// TwinCAT 3 PLC project PLC
// Title: Spreizanlage
// Company: fhnw
// ProjectVersion: 1.0.0.0
// ProgramVersion: 3.1.4026.14
// CompilerDefines: VISU_USEPROPERTYINFO
// libraries:
//   Tc2_MC2, * (Beckhoff Automation GmbH)
//   Tc2_Standard, * (Beckhoff Automation GmbH)
//   Tc2_System, * (Beckhoff Automation GmbH)
//   Tc2_TcpIp, * (Beckhoff Automation GmbH)
//   Tc2_Utilities, * (Beckhoff Automation GmbH)
//   VisuDialogs, * (System)
//   VisuSymbols, * (System)
// project tree:
//   DUTs/ ProcessData.TcDUT, State.TcDUT
//   / GlobalTextList.TcGTLO, PlcTask.TcTTO, Visualization Manager.TcVMO (not stored), VISU_TASK.TcTTO
//   GVLs/ GVL.TcGVL, GVL_Axis.TcGVL, GVL_HMI.TcGVL, GVL_Parameter.TcGVL
//   Lib/UDP/ FB_UDP_Connection.TcPOU, FB_UDP_ScanControl30x0.TcPOU
//   POUs/ FB_ControlPad.TcPOU, FB_FileWriter.TcPOU, FB_Izumi.TcPOU, FB_LaserScanner.TcPOU, FB_Winder.TcPOU, MAIN.TcPOU
//   VISUs/ GeneralSettings.TcVIS, MainWindow.TcVIS, Manual_Mode.TcVIS, Production_Mode.TcVIS, Setup_Mode.TcVIS, Winder_control.TcVIS
// real-time tasks:
//   TASK PlcTask: cycle T#10ms, priority 20, ADS port 350
//   TASK VisuTask: cycle T#200000us, priority 30, ADS port 351
// motion (NC):
//   TASK NC-Task 1 SAF: cycle T#2ms, priority 4, ADS port 501
//   TASK NC-Task 1 SVB: cycle T#10ms, priority 8, ADS port 511
//   AXIS Achse 1 (id 1)
//     General: UnitName=°
//     Dynamic: Acceleration=1592.706, Deceleration=1592.706, Jerk=4778.118
//     Velo: RefSearch=10.61804, RefSync=10.61804, SlowManual=53.0902, FastManual=318.5412, Fast=1061.804, Maximum=1061.804
//     OtherSettings: AllowMotionCmdToSlave=true
//     encoder EncType=19
//       EncPara: ScaleFactorNumerator=360, ScaleFactorDenominator=12582912, Inverse=true, MaxCount=#xffffffff
//     drive DrvType=16
//       DrvPara: Inverse=true, MaxCount=#xffffffff, DriveControlDWord=#x00020000
//         Analog: VeloReferenz=1167.9844, VeloScale=32, TorqueSetpointScale=10, ScaleFactorActTorque=0.1
//         TimeComp: TaskDelayCycles=1
//     controller CtrType=1
//       CtrPara: PriorControlFactor=1
//         Observer: BandWidth=20
// I/O:
//   DEVICE Gerät 1 (EtherCAT), AmsNetId 192.168.1.15.2.1
//     Klemme 1 (EK1100) [EK1100 EtherCAT-Koppler (2A E-Bus)]
//       Klemme 2 (EL1859) [EL1859 8K. Dig. Eingang 24V, 3ms, 8K. Dig. Ausgang 24V, 0.5A]
//       Klemme 3 (EL3064) [EL3064 4K.Ana. Eingang 0-10V]
//       Klemme 4 (ELM7221-0010) [ELM7221-0010 1K. Servo-Motor-Endstufe (48 V, 8 A RMS OCT)]
//         startup 32785:27 := E02E0000 // DRV Motor Settings Ch.1 / Motor speed limitation
//         startup 28688:3 := 08 // DRV Outputs Ch.1 / Modes of operation
//         startup 28688:16 := FF7F // DRV Outputs Ch.1 / Positive torque limit value
//         startup 28688:17 := FF7F // DRV Outputs Ch.1 / Negative torque limit value
//         startup 32784:87 := 64 // DRV Amplifier Settings Ch.1 / Position loop velocity feed forward gain
//         startup 32784:109 := 64000000 // DRV Amplifier Settings Ch.1 / Torque feed forward gain
//         startup 28688:11 := A00F // DRV Outputs Ch.1 / Torque limitation
//         startup 32784:19 := 2C02 // DRV Amplifier Settings Ch.1 / Current loop proportional gain
//         startup 32784:18 := 1500 // DRV Amplifier Settings Ch.1 / Current loop integral time
//         startup 32784:21 := 70000000 // DRV Amplifier Settings Ch.1 / Velocity loop proportional gain
//         startup 32784:20 := 96000000 // DRV Amplifier Settings Ch.1 / Velocity loop integral time
//       Klemme 5 (EL2634) [EL2634 4K. Relais Ausgang, Schließer (250 AC / 30V DC)]
//       Klemme 7 (EL9011) [EL9011 Endklemme]
//     Box 6 (NETX 51-RE/ECS) [NETX 51-RE/ECS]
// variable links:
//   NC-Task 1 SAF/Axes/Achse 1 <-> Device 1 (EtherCAT)/Term 1 (EK1100)/Term 4 (ELM7221-0010)
//     Drive/Inputs/In/nDataIn1 <-> DRV Following error actual value/Following error actual value
//     Drive/Inputs/In/nDataIn3[0] <-> DRV Torque actual value/Torque actual value
//     Drive/Inputs/In/nDcOutputTime <-> InfoData/DcOutputShift
//     Drive/Inputs/In/nState1 <-> DRV Statusword/Statusword
//     Drive/Inputs/In/nState2 <-> DRV Statusword/Statusword @bit 8
//     Drive/Inputs/In/nState4 @bit 1 <-> WcState/InputToggle
//     Drive/Inputs/In/nState4 <-> WcState/WcState
//     Drive/Outputs/Out/nCtrl1 <-> DRV Controlword/Controlword
//     Drive/Outputs/Out/nCtrl2 <-> DRV Controlword/Controlword @bit 8
//     Drive/Outputs/Out/nDataOut1 <-> DRV Target position/Target position
//     Drive/Outputs/Out/nDataOut2 <-> DRV Target velocity/Target velocity
//     Enc/Inputs/In/nDataIn1 <-> FB Position/Position
//     Enc/Inputs/In/nDcInputTime <-> InfoData/DcInputShift
//     Enc/Inputs/In/nState4 @bit 1 <-> WcState/InputToggle
//     Enc/Inputs/In/nState4 <-> WcState/WcState
//   PLC Instance <-> Device 1 (EtherCAT)/Term 1 (EK1100)/Term 2 (EL1859)
//     PlcTask Inputs/MAIN.ControlPad.bDigital_DecSpeed <-> Channel 5/Input
//     PlcTask Inputs/MAIN.ControlPad.bDigital_EStop <-> Channel 1/Input
//     PlcTask Inputs/MAIN.ControlPad.bDigital_IncSpeed <-> Channel 4/Input
//     PlcTask Inputs/MAIN.ControlPad.bDigital_Start <-> Channel 3/Input
//     PlcTask Inputs/MAIN.ControlPad.bDigital_Stop <-> Channel 2/Input
//   PLC Instance <-> Device 1 (EtherCAT)/Term 1 (EK1100)/Term 3 (EL3064)
//     PlcTask Inputs/MAIN.fbIzumi.iIzumiData <-> AI Standard Channel 1/Value
//   PLC Instance <-> NC-Task 1 SAF/Axes/Achse 1
//     PlcTask Inputs/MAIN.fbWinder.winderAxis.NcToPlc <-> Outputs/ToPlc
//     PlcTask Outputs/MAIN.fbWinder.winderAxis.PlcToNc <-> Inputs/FromPlc

CONFIGURATION PLC
    RESOURCE PLC ON TwinCAT3
        TASK PlcTask(INTERVAL := T#10ms, PRIORITY := 20);
        TASK VISU_TASK(INTERVAL := T#200000us, PRIORITY := 30);
        PROGRAM MAIN WITH PlcTask : MAIN;
        PROGRAM VisuElems_Visu_Prg WITH VISU_TASK : VisuElems.Visu_Prg;
    END_RESOURCE
END_CONFIGURATION

// ---- DUTs/ProcessData.TcDUT
TYPE ProcessData :
STRUCT
    Id          	: DINT;
    Value       	: DINT;
	RunningLength 	: REAL;  // Tape running length [m]
	Torque			: REAL; // Torque [?]
	TapeWidth		: REAL; // Measured width of tape (Laserscanner)
	LateralGap		: REAL;
	Airflow			: REAL;
	Temperature		: REAL;
    Timestamp   	: T_MaxString; 
END_STRUCT
END_TYPE

// ---- DUTs/State.TcDUT
{attribute 'qualified_only'}
{attribute 'strict'}
TYPE State :
(
	Error := 0,
	ManualMode,
	SetupMode,
	ProductionMode,
	ModusSelection
);
END_TYPE

// ---- GVLs/GVL.TcGVL
{attribute 'qualified_only'}
VAR_GLOBAL
	iTensionMonitoringData		: INT;		// in Newton [N]
	LaserScannerData : ARRAY[1..3] OF BYTE; // Testvariable für Laser Scanner Data
END_VAR

// ---- GVLs/GVL_Axis.TcGVL
{attribute 'qualified_only'}
VAR_GLOBAL
	// Winder Commands
	bCmdEnableWinder			: BOOL;
	bCmdStartWinder				: BOOL;
	bCmdStopWinder				: BOOL;
	bCmdResetWinder				: BOOL;
	
	// Winder Information
	bStatusPower				: BOOL;
	bStateCM					: BOOL;
	bStateStopping				: BOOL;
	bStateErrorStop				: BOOL;
	bNewMotionParameter			: BOOL;
	rWinderPos					: LREAL;
	
	// Winder Settings
	rWinderVelocity				: LREAL := 2.7;  // Speed reference value of winder [m/min]
	rWinderAcceleration			: LREAL := 1000;
	rWinderDeceleration			: LREAL := 1000;
	rWinderJerk					: LREAL := 1000;
	iWinderDirection			: INT := 1;
END_VAR

// ---- GVLs/GVL_HMI.TcGVL
{attribute 'qualified_only'}
VAR_GLOBAL
	bButtonWinderPower			: BOOL := TRUE;
	bButtonStartWinder			: BOOL;
	bButtonStopWinder			: BOOL;
	bButtonResetWinder			: BOOL;
	bButtonWinderDirection		: BOOL;
	bButtonNotWinderDirection	: BOOL;
	bButtonSelectionMode		: BOOL;
	bButtonSetupMode			: BOOL;
	bButtonManualMode			: BOOL;
	bButtonProdutionMode 		: BOOL;
	ActTapeSpeed				: REAL;
	ActTorque					: LREAL;
	RunningLength				: REAL;
END_VAR

// ---- GVLs/GVL_Parameter.TcGVL
{attribute 'qualified_only'}
VAR_GLOBAL PERSISTENT  // Parameters are PERSISTENT --> Parameter will remain stored
	Offset_Izumi  				: INT := 0; // Zur Kalibration der Izumi Daten
	EmptySpoolDiameter 			: REAL:=100; // Diameter of the spool [mm] (used to calculate required motor speed) 
	SpeedChange 				: LREAL := 0.2; // Increment/Decrement of speed ref. whenever control pad is used [m/min]
	tMeas_SetupMode 			: REAL := 500;  // measuring cycle time in manual mode [ms]
	tMeas_ProductionMode 		: REAL := 1000;  // measuring cycle time in prod. mode [ms]
	TapeHeight					: REAL := 0.1;  // Used to adjust speed refence with increasing spool diameter [mm]
	rWinderAcceleration			: LREAL;
	rWinderDeceleration			: LREAL;
	rWinderJerk					: LREAL;
END_VAR

// ---- POUs/MAIN.TcPOU
PROGRAM MAIN
VAR
	fbWinder			: FB_Winder;
	fbIzumi				: FB_Izumi;
	fbLaserScanner		: FB_LaserScanner;
	ActualState			: State := State.ManualMode;
	ControlPad			: FB_ControlPad;
	StartWinder			: BOOL;   // Cmd. to start winder
	StartWinder_prev	: BOOL; // For edge detection
	StopWinder			: BOOL;   // Cmd. to stop winder
	
	fbTime   			: FB_LocalSystemTime := ( bEnable := TRUE, dwCycle := 1 );  // System time synchronization 
	logTimer 			: TON := ( IN := TRUE, PT := T#500MS );  // Timer used to generate the data acq. trigger pulse
	fbWriteFile     	: FB_FileWriter;
	arrTestData     	: ARRAY[0..10] OF ProcessData;
    nIteration      	: INT;
    bStartNewJob    	: BOOL;
    fbFormatString  	: FB_FormatString;
	fbGetCurrentTaskIndex   : GETCURTASKINDEX;
	tStorage			: TIME := T#1000MS;  // frequency of data acquistion (mode dependent) [Hz]
	FileCnt				: UINT := 0;
	FileCnt_prev		: UINT := 0;
	FileName				: STRING := '00';
	// Variablen für LaserScanner
	//fbSocketCloseAll	: FB_SocketCloseAll;
	//fbUDP_ScanControl	: FB_UDP_ScanControl30x0;
	//Connect : BOOL := TRUE; // True = Verbindung aktiv
	//TestSend : BOOL; // Test send bit
	//Res : BOOL;
END_VAR
VAR CONSTANT
	cHeader 			: STRING := 'Time stamp;ID;Value;Airflow [l/min];Running Length [m];$n';
END_VAR

(*
Beispiel der UDP Verbindung zum LaserScanner  --> Kopie des Beispielprojektes.

Anforderungen:
1. Auf der IPC muss das Packet TF6310 installiert sein
2. Im Projekt muss die Lizenz TF6310 ausgewählt sein
3. SocketCloseAll muss zu Begin ins Projekt eingebaut werden
   (Schliesst alle offenen Sockets => Aufräumen)
*)
(*
fbSocketCloseAll(bExecute := TRUE);

fbUDP_ScanControl(
	Enable:= NOT fbSocketCloseAll.bBusy AND Connect, 
	LocalHost:= '192.168.50.10', 
	LocalPort:= 61000, 
	SocketCreated=> , 
	ConnectionBusy=> , 
	ConnectionError=> );
	
IF TestSend THEN
	TestSend := FALSE;
	Res := fbUDP_ScanControl.SendString('Das ist ein Test', '192.168.111.1\n', 20000);
END_IF
*)
fbTime();

(* State Machine (Modus selection) *)
CASE ActualState OF
	State.ModusSelection:
	// Kommandos TO BE DONE

		IF GVL_HMI.bButtonSetupMode THEN
			ActualState := State.SetupMode;
		ELSIF GVL_HMI.bButtonManualMode THEN
			ActualState := State.ManualMode;
		ELSIF GVL_HMI.bButtonProdutionMode THEN
			ActualState := State.ProductionMode;
		END_IF
	State.ManualMode:
	// Kommandos TO BE DONE
		IF GVL_HMI.bButtonSetupMode THEN
			ActualState := State.SetupMode;
		ELSIF GVL_HMI.bButtonSelectionMode THEN
			ActualState := State.ModusSelection;
		ELSIF GVL_HMI.bButtonProdutionMode THEN
			ActualState := State.ProductionMode;
		END_IF
	State.ProductionMode:
		// Kommandos TO BE DONE
		logTimer.PT := TO_TIME(GVL_Parameter.tMeas_ProductionMode);  // measuring freq. [Hz]
		IF GVL_HMI.bButtonSetupMode THEN
			ActualState := State.SetupMode;
		ELSIF GVL_HMI.bButtonManualMode THEN
			ActualState := State.ManualMode;
		ELSIF GVL_HMI.bButtonSelectionMode THEN
			ActualState := State.ModusSelection;
		END_IF
	State.SetupMode:
		// Kommandos TO BE DONE
		logTimer.PT := TO_TIME(GVL_Parameter.tMeas_SetupMode);  // measuring freq. [Hz]
		IF GVL_HMI.bButtonSelectionMode THEN
			ActualState := State.ModusSelection;
		ELSIF GVL_HMI.bButtonManualMode THEN
			ActualState := State.ManualMode;
		ELSIF GVL_HMI.bButtonProdutionMode THEN
			ActualState := State.ProductionMode;
		END_IF
		
END_CASE


// ----------------- Laser Scanner ------------------------
fbLaserScanner();
GVL.LaserScannerData := fbLaserScanner.DataOut;	

StartWinder := GVL_Axis.bCmdStartWinder OR ControlPad.StartCmd;
StopWinder := GVL_Axis.bCmdStopWinder OR ControlPad.StopCmd;

IF fbWinder.bStateCM THEN
	ControlPad.En_SpeedRefChg := TRUE;
ELSE
	ControlPad.En_SpeedRefChg := FALSE;
END_IF

// MC Winder
fbWinder(
	bEnableWinder			:= GVL_Axis.bCmdEnableWinder,
	bStartWinder			:= StartWinder,
	bStopWinder				:= StopWinder,
	bResetWinder			:= GVL_Axis.bCmdResetWinder,
	VelocityRef				:= GVL_Axis.rWinderVelocity + ControlPad.AddSpeed,
	bStatusPower			=> GVL_Axis.bStatusPower,
	bStateCM				=> GVL_Axis.bStateCM,
	bStateStopping			=> GVL_Axis.bStateStopping,
	bStateErrorStop			=> GVL_Axis.bStateErrorStop,
	bNewMotionParameter		=> GVL_Axis.bNewMotionParameter,
	ActTapeSpeed			=> GVL_HMI.ActTapeSpeed,
	ActualTorque_Nm			=> GVL_HMI.ActTorque,
	RunningLength			=> GVL_HMI.RunningLength);								
	
// Izumi Data
fbIzumi(
	iIzumiInNewton			=> GVL.iTensionMonitoringData);
	
// Control Pad
ControlPad();
	
// HMI Configuration
GVL_Axis.bCmdEnableWinder	:= GVL_HMI.bButtonWinderPower;
GVL_Axis.bCmdStartWinder	:= GVL_HMI.bButtonStartWinder;
GVL_Axis.bCmdStopWinder		:= GVL_HMI.bButtonStopWinder;
GVL_Axis.bCmdResetWinder	:= GVL_HMI.bButtonResetWinder;

IF GVL_HMI.bButtonWinderDirection THEN
	GVL_Axis.iWinderDirection := 3;			// Counter-Clockwise/Negative Direction
ELSE
	GVL_Axis.iWinderDirection := 1;			// Clockwise/Positive Direction
END_IF
GVL_HMI.bButtonNotWinderDirection := NOT GVL_HMI.bButtonWinderDirection;

// ----------------- Schreiben der Daten (https://stackoverflow.com/questions/76112520/how-do-i-save-data-from-my-plc-in-excel-or-csv-format-in-twincat) ------------------
// Trigger data acq. acc. to desired measuring freq.
IF StartWinder AND NOT(StartWinder_prev) THEN
	FileCnt := FileCnt+1;
	FileName := SYSTEMTIME_TO_STRING(fbTime.systemTime);
END_IF
StartWinder_prev := StartWinder;

fbWriteFile(
	//sFileName   := CONCAT(CONCAT('Measurement_',TO_STRING(FileCnt)),'.csv'),
	sFileName   := CONCAT(TO_STRING(FileCnt),'.csv'),
    sFilePath   := 'C:\',
    sNetId      := '');

IF FileCnt_prev <> FileCnt THEN
	fbWriteFile.WriteToFile(message := cHeader);
END_IF

FileCnt_prev := FileCnt;

	(*NewFileName := CONCAT(NewFileName,'-');
	NewFileName := CONCAT(NewFileName,WORD_TO_STRING(fbTime.systemTime.wMonth));
	NewFileName := CONCAT(NewFileName,'-');
	NewFileName := CONCAT(NewFileName,WORD_TO_STRING(fbTime.systemTime.wYear));
	NewFileName := CONCAT(NewFileName,'_at_');
	NewFileName := CONCAT(NewFileName,WORD_TO_STRING(fbTime.systemTime.wHour));
	NewFileName := CONCAT(NewFileName,'-');
	NewFileName := CONCAT(NewFileName,WORD_TO_STRING(fbTime.systemTime.wMinute));
	NewFileName := CONCAT(NewFileName,'-');
	NewFileName := CONCAT(NewFileName,WORD_TO_STRING(fbTime.systemTime.wSecond));*)

(*fbGetCurrentTaskIndex();
IF _TaskInfo[fbGetCurrentTaskIndex.index].FirstCycle THEN
    fbWriteFile.WriteToFile(message := cHeader);
END_IF*)

logTimer( IN := fbTime.bValid AND fbWinder.bStateCM);  // Start trigger for data acq.
IF logTimer.Q THEN
    logTimer( IN := FALSE );
	logTimer( IN := fbTime.bValid );
	bStartNewJob := TRUE;
END_IF

IF bStartNewJob THEN
    // Making up some fake data to store it
    arrTestData[nIteration].Id := nIteration;                   // just some made up id
    arrTestData[nIteration].Value := 5*nIteration;              // just some made up value
	arrTestData[nIteration].Airflow := 23.6;
	arrTestData[nIteration].RunningLength := fbWinder.RunningLength;
    arrTestData[nIteration].Timestamp := SYSTEMTIME_TO_STRING(fbTime.systemTime); 
    
    // Create the full line by using the FB_FormatString, way easier than CONCAT
    fbFormatString(
        sFormat := '%s;%d;%d;%f;%f$n',
		arg1    := F_STRING(arrTestData[nIteration].Timestamp),
        arg2    := F_DINT(arrTestData[nIteration].Id),
        arg3    := F_DINT(arrTestData[nIteration].Value),
		arg4	:= F_REAL(arrTestData[nIteration].Airflow),
		arg5	:= F_REAL(arrTestData[nIteration].RunningLength));

    // Send the created line to the file writer
    fbWriteFile.WriteToFile(message := fbFormatString.sOut);

    // Increasing the counter for new, different data
    IF nIteration <10 THEN
        nIteration := nIteration + 1;
    ELSE
        nIteration := 0;
    END_IF
    
    // And finally, clear the trigger
    bStartNewJob := FALSE;      
END_IF

END_PROGRAM

// ---- POUs/FB_Winder.TcPOU
FUNCTION_BLOCK FB_Winder
VAR_INPUT
	bEnableWinder			: BOOL;
	bStartWinder			: BOOL;
	bStopWinder				: BOOL;
	bResetWinder			: BOOL;
	VelocityRef				: REAL;
	bCountRev				: BOOL; // IF TRUE revolutions will be counted
END_VAR
VAR_OUTPUT
	bStatusPower			: BOOL;
	bStateCM				: BOOL;
	bStateStopping			: BOOL;
	bStateErrorStop			: BOOL;
	bNewMotionParameter		: BOOL;
	bStateError				: BOOL; // Drive indicates an error
	ErrorCode				: UDINT; // Error code received from drive
	RevCounter				: DINT; // Revolution counter --> required for speed ref. calculation
	ActTapeSpeed			: REAL; // Act. tape speed [m/min]
	RunningLength			: REAL; // Act. running length [m]
	ActualTorque_Nm			: LREAL; // Actual motor torque [Nm]
END_VAR
VAR
	fbWinderStatus			: MC_ReadStatus;
	fbReset					: MC_Reset;
	fbWinderPower			: MC_Power;
	fbWinderMV				: MC_MoveVelocity;
	fbWinderStop			: MC_Stop;
	fbWinderReset			: MC_Reset;
	winderAxis				: AXIS_REF;
	refvelocity				: LREAL;
	refvelocity_prev		: LREAL := 0.0; // to detect speed ref, changes
END_VAR

(* ------------ Calculate speed reference value from tape speed ---------------
vref = refvelocity [°/s]
vtape = tape speed [m/min]
d_spool = diameter of spool [mm]
vref = 
*)
//refvelocity := GVL_Axis.rWinderVelocity*6000/(PI*GVL_Parameter.EmptySpoolDiameter); // m/min --> °/s

refvelocity := VelocityRef*6000/(PI*GVL_Parameter.EmptySpoolDiameter); // m/min --> °/s

// ------------ MC_ReadStatus ------------
fbWinderStatus(
	Axis			:= winderAxis,
	Enable			:= TRUE);
	
	
bStateCM			:= fbWinderStatus.ContinuousMotion;
bStateStopping		:= fbWinderStatus.Stopping;
bStateErrorStop		:= fbWinderStatus.ErrorStop;
bStateError 		:= fbWinderStatus.Error;
ErrorCode	 		:= fbWinderStatus.ErrorID;


fbReset(Axis := winderAxis, Execute := bStateError);
fbReset(Axis := winderAxis, Execute := FALSE);

// ------------ MC_Power ------------
IF bEnableWinder THEN
	fbWinderPower(
		Axis			:= winderAxis,
		Enable			:= TRUE,
		Enable_Positive	:= TRUE,
		Enable_Negative	:= TRUE);
ELSE
	fbWinderPower(
		Axis			:= winderAxis,
		Enable			:= FALSE);
END_IF
bStatusPower		:= fbWinderPower.Status;

// ------------ MC_MoveVelocity ------------
//IF (bStartWinder AND fbWinderStatus.Status.NotMoving) OR ((refvelocity <> refvelocity_prev) AND fbWinderStatus.Status.ContinuousMotion) THEN
IF (bStartWinder) OR ((refvelocity <> refvelocity_prev)) THEN
	RunningLength := 0.0;  // Reset calculated running length whenever restarting
	fbWinderMV(
		Axis			:= winderAxis,
		Execute			:= TRUE,
		Velocity		:= refvelocity,
		Acceleration	:= GVL_Axis.rWinderAcceleration,
		Deceleration	:= GVL_Axis.rWinderDeceleration,
		Jerk			:= GVL_Axis.rWinderJerk,
		Direction		:= GVL_Axis.iWinderDirection);
	refvelocity_prev 	:= refvelocity;
ELSE
	fbWinderMV(
		Axis			:= winderAxis,
		Execute			:= FALSE);
END_IF

// Not sure whta this is supposed to be used for --> currently it only triggers an text indication on the Visu
IF fbWinderMV.Velocity <> GVL_Axis.rWinderVelocity OR
   fbWinderMV.Acceleration <> GVL_Axis.rWinderAcceleration OR
   fbWinderMV.Deceleration <> GVL_Axis.rWinderDeceleration OR
   fbWinderMV.Jerk <> GVL_Axis.rWinderJerk OR
   fbWinderMV.Direction <> GVL_Axis.iWinderDirection THEN
	bNewMotionParameter	:= TRUE;
ELSE
	bNewMotionParameter	:= FALSE;
END_IF

// ------------ MC_Stop ------------
IF bStopWinder THEN
	fbWinderStop(
		Axis			:= winderAxis,
		Execute			:= TRUE);
ELSE
	fbWinderStop(
		Axis			:= winderAxis,
		Execute			:= FALSE); 
END_IF

// ------------ MC_Reset ------------
IF bResetWinder THEN
	fbWinderReset(
		Axis			:= winderAxis,
		Execute			:= TRUE);
ELSE
	fbWinderReset(
		Axis			:= winderAxis,
		Execute			:= FALSE);
END_IF

// ------------- Calculate no. of revolutions ---------------
IF bCountRev THEN
	RevCounter := ABS(winderAxis.NcToPlc.ModuloActTurns); 
ELSE
	RevCounter := 0;
END_IF

(* ------------- Calculate actual tape related values ----------------
vtape = tape speed [m/min]
vact = actual motor speed [°/s]
dspool = diameter of spool [mm]
nact = (vact*PI/180°)/(2*PI) = vact/360  (angular velocity/ (2*PI))
vtape = nact *(PI*dspool) = vact*PI*dspool/360 * (60s/min)/(1000mm/m) = vact*PI*dspool/6000
*)
ActTapeSpeed := TO_REAL(ABS(winderAxis.NcToPlc.ActVelo) * PI * GVL_Parameter.EmptySpoolDiameter)/6000; // °/s --> m/min
RunningLength := RunningLength + ActTapeSpeed * 0.01 / 60; // Integrate TapeSpeed (important: Task cycle time needs to be adapted whenever modified)
ActualTorque_Nm := winderAxis.NcToPlc.ActTorque/10;  // Actual torque [?] --> ToDo: Check internal scaling

END_FUNCTION_BLOCK

// ---- POUs/FB_Izumi.TcPOU
FUNCTION_BLOCK FB_Izumi
VAR_INPUT
END_VAR
VAR_OUTPUT
	iIzumiInNewton			: INT;	// converted to Newton
END_VAR
VAR
	iIzumiData AT %I* 		: INT;	// measured in mV
	iVoltage AT %I* 		: INT;	// Voltage sensor
END_VAR

iIzumiInNewton 				:= iIzumiData/100;

END_FUNCTION_BLOCK

// ---- POUs/FB_LaserScanner.TcPOU
FUNCTION_BLOCK FB_LaserScanner
VAR_INPUT
END_VAR
VAR_OUTPUT
	Error,Busy,SocketCreated : BOOL; //Status indication
	DataOut : ARRAY[1..3] OF BYTE;
END_VAR
VAR
	fbSocketCloseAll	: FB_SocketCloseAll;
	fbUDP_ScanControl	: FB_UDP_ScanControl30x0;
	Connect : BOOL := TRUE; // True = Verbindung aktiv
	TestSend : BOOL; // Test send bit
	Res : BOOL;
END_VAR

(*
Beispiel der UDP Verbindung zum LaserScanner  --> Kopie des Beispielprojektes.

Anforderungen:
1. Auf der IPC muss das Packet TF6310 installiert sein
2. Im Projekt muss die Lizenz TF6310 ausgewählt sein
3. SocketCloseAll muss zu Begin ins Projekt eingebaut werden
   (Schliesst alle offenen Sockets => Aufräumen)
*)
fbSocketCloseAll(bExecute := TRUE);

fbUDP_ScanControl(
	Enable:= NOT fbSocketCloseAll.bBusy AND Connect, 
	LocalHost:= '192.168.50.10', 
	LocalPort:= 61000, 
	SocketCreated=> SocketCreated, 
	ConnectionBusy=> Busy, 
	ConnectionError=> Error,
	DataOut=> DataOut);
	
IF TestSend THEN
	TestSend := FALSE;
	Res := fbUDP_ScanControl.SendString('Das ist ein Test', '192.168.111.1\n', 20000);
END_IF

END_FUNCTION_BLOCK

// ---- Lib/UDP/FB_UDP_ScanControl30x0.TcPOU
/// Implementierung für ScanControl 30x0
FUNCTION_BLOCK FB_UDP_ScanControl30x0 EXTENDS FB_UDP_Connection
VAR_INPUT
END_VAR
VAR_OUTPUT
	DataOut : ARRAY[1..3] OF BYTE;
END_VAR
VAR
	Data : ARRAY[0..5000] OF BYTE;
	DataString : STRING(5000);
	Value1 : INT;
	Value2 : INT;
	Value3 : INT;
	Value4 : INT;
	Value5 : DINT;
	Test : ARRAY[1..3] OF BYTE;
END_VAR

// Aufruf des Body der Basisklasse
SUPER^();

METHOD PROTECTED OnNewMessage
VAR_INPUT
	pData	: POINTER TO BYTE;
	DataLen	: UDINT;
END_VAR
VAR
	
END_VAR
(*
Diese Methode ist überschrieben aus der Basisklasse
Bei einer eingehenden Meldung, können die DAten hier geparst und verarbeitet werden.
*)

// Demo
MEMSET(ADR(Data), 0, SIZEOF(Data)); // Speicherbereich leeren
MEMCPY(ADR(Data), pData, DataLen);  // 
MEMSET(ADR(DataString),0, SIZEOF(DataString));
MEMCPY(ADR(DataString), pData, DataLen);

MEMCPY(ADR(DataOut), pData, 3);
END_METHOD

END_FUNCTION_BLOCK

// ---- Lib/UDP/FB_UDP_Connection.TcPOU
/// Basis Baustein für das erstellen einer UDP Verbindung
FUNCTION_BLOCK FB_UDP_Connection
VAR_INPUT
	Enable					: BOOL; // True = Verbindung herstellen
	LocalHost				: T_IPv4Addr := '0.0.0.0'; // Lokale Adresse 
	LocalPort				: UDINT; // Lokaler Port
END_VAR
VAR_OUTPUT
	SocketCreated			: BOOL; // UDP Socket erstellt
	ConnectionBusy			: BOOL; // UDP Socket-Erstellung läuft
	ConnectionError			: BOOL; // UDP Socket-Erstellung Fehler
	SendBusy				: BOOL; // Senden im gange
END_VAR
VAR
	(* Receive Buffer
	   Wird eine Grösse über 8100 Byte benötigt, 
	   Paramter in der Globalen Variablenliste anpassen:
	   TCPADS_MAXUDP_BUFFSIZE
	*)
	ReceiveBuffer			: ARRAY[0..BUFFER_SIZE] OF BYTE;
	fbReceiveFrom			: FB_SocketUdpReceiveFrom;
	fbSendTo				: FB_SocketUdpSendTo;
	fbConnectionLessSocket 	: FB_ConnectionlessSocket;
END_VAR
VAR CONSTANT
	BUFFER_SIZE 			: DINT := 2000; // Data Buffer in Byte
END_VAR

// Dieser Baustein erstellt ein Socket
fbConnectionLessSocket(
	nMode := 0,
	sLocalHost := LocalHost,
	nLocalPort := LocalPort,
	bEnable := Enable,
	bBusy => ConnectionBusy,
	bError => ConnectionError);

SocketCreated := fbConnectionLessSocket.eState = E_SocketConnectionlessState.eSOCKET_CREATED;

// Daten empfangen
// -----------------------
fbReceiveFrom(
	sSrvNetId:= , 
	hSocket:= fbConnectionLessSocket.hSocket, 
	cbLen:= SIZEOF(ReceiveBuffer),
	pDest:= ADR(ReceiveBuffer),
	bExecute:= SocketCreated AND NOT fbReceiveFrom.bBusy, 
	tTimeout:= , 
	bBusy=> , 
	bError=> , 
	nErrId=> , 
	sRemoteHost=> , 
	nRemotePort=> , 
	nRecBytes=> );
	
IF NOT fbReceiveFrom.bBusy THEN
	IF fbReceiveFrom.nRecBytes > 0 THEN
		// Anzahl 
		OnNewMessage(ADR(ReceiveBuffer), fbReceiveFrom.nRecBytes);
	END_IF
END_IF

// Daten senden
// Wird über die Methode Send() resp. SendString() getriggert.
// Aufruf nötigt bis Message gesendet ist
// -------------------------------------
fbSendTo(
	bBusy=> SendBusy, 
	bError=> , 
	nErrId=> );

/// Callback Methode bei eingegangenen Daten
METHOD PROTECTED OnNewMessage
VAR_INPUT
	pData	: POINTER TO BYTE; // Pointer zu den eingegangenen Daten
	DataLen	: UDINT; // Datenlänge
END_VAR
(*
Diese Methode kann in einer vererbten Klasse überschrieben werden, 
um den Basis Code nicht mit dem Prozess zu binden
*)
;
END_METHOD

/// Senden von Daten
METHOD Send : BOOL // True = Senden erfolgreich getriggert
VAR_INPUT
	pData		: POINTER TO BYTE; // Trigger tu den Daten
	DataLen		: UDINT; // Datenlänge
	RemotePeer 	: T_IPv4Addr; // Ziel Host
	RemotePort 	: UDINT; // Ziel Port
END_VAR

IF fbSendTo.bBusy OR NOT SocketCreated THEN
	Send := FALSE;
	RETURN;
END_IF


fbSendTo(
	bExecute := TRUE,
	hsocket := fbConnectionLessSocket.hSocket,
	sRemoteHost := RemotePeer,
	nRemotePort := RemotePort,
	cbLen := DataLen,
	pSrc := pData,
	bBusy => SendBusy);
	
fbSendTo(bExecute := FALSE);

Send := NOT fbSendTO.bError;
END_METHOD

/// Senden eines Strings
METHOD SendString : BOOL // True = Erfolgreich getriggert
VAR_IN_OUT CONSTANT
	Data	: STRING; // String Daten
END_VAR
VAR_INPUT
	RemotePeer 	: T_IPv4Addr; // Ziel Adresse
	RemotePort 	: UDINT; // Ziel Port
END_VAR

IF LEN2(ADR(data)) = 0 THEN
	SendString := FALSE;
	RETURN;
END_IF

SendString := Send(
				pData := ADR(Data),
				DataLen := LEN2(ADR(Data)),
				RemotePeer := RemotePeer,
				RemotePort := RemotePort);
END_METHOD

END_FUNCTION_BLOCK

// ---- POUs/FB_ControlPad.TcPOU
FUNCTION_BLOCK FB_ControlPad
VAR_INPUT
	Reset 			: BOOL;
	En_SpeedRefChg 	: BOOL;  // Only when enebaled speed inc./dec. will be possible
END_VAR
VAR_OUTPUT
	EStopLatch	: BOOL;
	StartCmd	: BOOL;  // Start Cmd. Trigger
	StopCmd 	: BOOL;  // Stop Cmd. trigger
	AddSpeed    : LREAL := 0.0; // Speed Offset to actual speed
END_VAR
VAR
	bDigital_EStop AT %I* 		: BIT;	
	bDigital_Start AT %I* 		: BIT;
	bDigital_Stop AT %I* 		: BIT;
	bDigital_IncSpeed AT %I*	: BIT;
	bDigital_DecSpeed AT %I*	: BIT;
	IncSpeed_prev				: BIT;
	DecSpeed_prev				: BIT;
	Start_prev					: BIT := FALSE;  // for edge detection
	Stop_prev					: BIT := FALSE;  // for edge detection
END_VAR

IF NOT(bDigital_EStop) THEN
	EStopLatch := TRUE; // Latch E-Stop for indication
END_IF

IF EStopLatch AND Reset THEN // Reset Latched signal for indication
	EStopLatch := FALSE;
END_IF

// -------- Start Cmd. trigger to start motor (edge detection) --------
IF bDigital_Start AND NOT(Start_prev) THEN
	StartCmd := TRUE;
ELSE
	StartCmd := FALSE;
END_IF
Start_prev := bDigital_Start;

// -------- Stop Cmd. trigger to stop motor (edge detection) --------
IF bDigital_Stop AND NOT(Stop_prev) THEN
	StopCmd := TRUE;
ELSE
	StopCmd := FALSE;
END_IF
Stop_prev := bDigital_Stop;

// Speed ref. offset value created by Control pad
IF En_SpeedRefChg THEN
	IF bDigital_IncSpeed AND NOT(IncSpeed_prev) THEN
		AddSpeed := AddSpeed + GVL_Parameter.SpeedChange;
	ELSIF bDigital_DecSpeed AND NOT(DecSpeed_prev) THEN
		AddSpeed := AddSpeed - GVL_Parameter.SpeedChange;
	END_IF
	IncSpeed_prev := bDigital_IncSpeed;
	DecSpeed_prev := bDigital_DecSpeed;
ELSE
	AddSpeed := 0.0;
END_IF

END_FUNCTION_BLOCK

// ---- POUs/FB_FileWriter.TcPOU
FUNCTION_BLOCK FB_FileWriter
VAR_INPUT
    sFilePath   : T_MaxString;
    sFileName   : T_MaxString;
    sNetId      : STRING;   // NetId of the target, leave empty for local
END_VAR
VAR
    fbFileOpen  : FB_FileOpen;
    fbFilePuts  : FB_FilePuts;
    fbFileClose : FB_FileClose;
    nFileHandle : UINT;
    
    arrBuffer   : ARRAY[0..100] OF T_MaxString;
    eFileWriteState : (IDLE, OPEN_FILE, WRITE_TO_FILE, CLOSE_FILE, ERROR);
END_VAR

CASE eFileWriteState OF
    IDLE:
        // Make sure all the file writing FBs are ready for use (trigger on execute)
        Init();
        
        // We have pending data to be written
        IF arrBuffer[0] <> '' THEN
            eFileWriteState := OPEN_FILE;
        END_IF
        
    OPEN_FILE:
        // Opens a file for writing at the end of the file (append). 
        // If the file does not exist, a new file is created.
        fbFileOpen(
            bExecute    := TRUE,
            sNetId      := sNetId,
            sPathName   := CONCAT(sFilePath, sFileName),
            nMode       := FOPEN_MODEAPPEND);
            
        IF fbFileOpen.bError THEN
            eFileWriteState := ERROR;
        ELSIF NOT fbFileOpen.bBusy THEN
            nFileHandle := fbFileOpen.hFile;
            fbFileOpen(bExecute := FALSE);
            eFileWriteState := WRITE_TO_FILE;
        END_IF
    
    WRITE_TO_FILE:
        fbFilePuts(
            bExecute    := TRUE,
            sNetId      := sNetId,
            hFile       := nFileHandle,
            sLine       := arrBuffer[0]);
        IF fbFilePuts.bError THEN
            eFileWriteState := ERROR;
        ELSIF NOT fbFileClose.bBusy THEN
            // Sucess, data was written
            // Rotate the buffer and close the file
            RotateBuffer();
            eFileWriteState := CLOSE_FILE; 
        END_IF
    
    CLOSE_FILE:
        fbFileClose(
            bExecute := TRUE,
            sNetId      := sNetId,
            hFile       := nFileHandle);
            
        IF fbFileClose.bError THEN
            eFileWriteState := ERROR;
        ELSIF NOT fbFileClose.bBusy THEN
            nFileHandle := 0;
            eFileWriteState := IDLE;
        END_IF      
    
    ERROR:
        // Error, clear the handle and go back to idle
        nFileHandle := 0;
        eFileWriteState := IDLE;
END_CASE

METHOD PRIVATE Init : BOOL
VAR_INPUT
END_VAR
fbFileClose(bExecute := FALSE);
fbFileOpen(bExecute := FALSE);
fbFilePuts(bExecute := FALSE);
END_METHOD

METHOD PRIVATE InsertToBuffer
VAR_INPUT
    value   : STRING;
END_VAR
VAR
    nBufferIndex    : INT;
END_VAR
FOR nBufferIndex := 0 TO 100 BY 1 DO
    IF arrBuffer[nBufferIndex] = '' THEN
        // We found the free spot in the buffer, insert the value to this place
        arrBuffer[nBufferIndex] := value;
        EXIT;
    END_IF
END_FOR
END_METHOD

METHOD PRIVATE RotateBuffer
VAR
    nIndex  : int := 0;
END_VAR
FOR nIndex := 0 TO 99 BY 1 DO
    // We can exit when we reached the empty slot in the buffer
    IF arrBuffer[nIndex] = '' THEN
        EXIT;
    END_IF
    // FIFO, removing first element in the array copying the next, etc...
    arrBuffer[nIndex] := arrBuffer[nIndex+1];
END_FOR
END_METHOD

METHOD WriteToFile : BOOL
VAR_INPUT
    message : T_MaxString;
END_VAR
InsertToBuffer(value := message);
END_METHOD

END_FUNCTION_BLOCK

// ---- GlobalTextList.TcGTLO
TEXTLIST GlobalTextList
  543 = "!!New Motion Parameter detected!!\nClick 'Start winder' to update Parameters"
  193 = '%2.2f'
  232 = '%5.0f'
  503 = '%5.1f'
  237 = '%5.2f'
  974 = '%6.1f'
  341 = '%f'
  431 = '%i'
  756 = 'Actual Motor Torque [%]'
  883 = 'Actual Motor Torque [Nm]'
  674 = 'Actual:'
  471 = 'Air flow [l/min]'
  186 = 'Air temp. [°C]'
  763 = 'Allows manual control (start/stop) of each and every subsystem.'
  842 = 'Allows to adjust general system parameters, which will be applied in all different modes of operation.'
  407 = 'Back to Main window'
  3 = 'Back to Main Window'
  227 = 'Clockwise'
  282 = 'Counter-\nClockwise'
  936 = 'Defines how often measurements will be taken and written to a file. Lower values will increase the file size.'
  686 = 'Drive speed [m/min]'
  441 = 'Empty Spool diameter [mm]:'
  397 = 'fan'
  905 = 'General settings'
  913 = 'Invert Winder\nDirection'
  607 = 'Main Window'
  430 = 'Manual Mode'
  119 = 'Manual Mode:'
  713 = 'Meas. cycle Prod. mode [ms]:'
  856 = 'Meas. cycle Setup mode [ms]:'
  881 = 'Measurement frequency:'
  170 = 'Moving'
  647 = 'Offset [N]:'
  608 = 'Operation mode supposed to be used for production with slightly reduced measurement frequency.'
  605 = 'Operation mode with increased measuring frequency in order to fine tune the process (e.g. reference values) according to your needs.'
  649 = 'Power up Winder'
  884 = 'Production Mode'
  987 = 'Reference:'
  614 = 'Required to calculate speed reference value for winder motor.'
  125 = 'Reset'
  156 = 'Reset needed'
  784 = 'Running length [m]'
  895 = 'Sensor Data'
  127 = 'Set:'
  289 = 'Setup Mode'
  333 = 'Speed Inc./Dec. [m/min]'
  327 = 'Speed increment and decrement applied using the control pad.'
  990 = 'Start winder'
  697 = 'Start winder with \nparameters'
  212 = 'STOP'
  577 = 'Stop winder'
  460 = 'Stopping'
  457 = 'Tape height [mm]'
  640 = 'tape width [mm]'
  247 = 'Tension Monitoring System\nOutput in Newton [N]'
  197 = 'Tension settings'
  835 = 'tow brake [g]'
  226 = 'tow tension [N]'
  516 = 'Winder Acceleration'
  509 = 'Winder control'
  633 = 'Winder Deceleration'
  721 = 'Winder Jerk'
  976 = 'Winder Power ON/OFF'
  663 = 'Winder settings'
  432 = 'Winder Velocity [m/min]'
END_TEXTLIST

// ---- VISUs/GeneralSettings.TcVIS
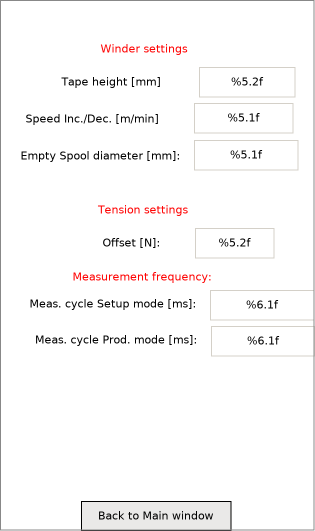
VISUALIZATION GeneralSettings  // 315x531
    Rectangle (81,501 150x30), "Back to Main window"
        OnMouseClick: change screen: MainWindow
    Textfield (199,67 96x30), "%5.2f", text variable: GVL_Parameter.TapeHeight
    Label (42,67 122x30), "Tape height [mm]"
    Label (69,34 150x30), "Winder settings"
    Textfield (194,103 99x30), "%5.1f", tooltip "Speed increment and decrement applied using the control pad.", text variable: GVL_Parameter.SpeedChange
        OnMouseClick: write GVL_Parameter.SpeedChange via VisuDialogs.Numpad
    Label (16,104 146x30), "Speed Inc./Dec. [m/min]"
    Textfield (195,228 79x30), "%5.2f"
    Label (41,228 122x30), "Offset [N]:"
    Label (68,195 150x30), "Tension settings"
    Textfield (194,140 104x30), "%5.1f", tooltip "Required to calculate speed reference value for winder motor.", text variable: GVL_Parameter.EmptySpoolDiameter
        OnMouseClick: write GVL_Parameter.EmptySpoolDiameter via VisuDialogs.Numpad, min 10, max 1000
    Label (16,141 167x30), "Empty Spool diameter [mm]:"
    Textfield (210,290 104x30), "%6.1f", tooltip "Defines how often measurements will be taken and written to a file. Lower values will increase the file size.", text variable: GVL_Parameter.tMeas_SetupMode
        OnMouseClick: write GVL_Parameter.tMeas_SetupMode via VisuDialogs.Numpad, min 10, max 100000, format 1000
    Label (14,289 185x30), "Meas. cycle Setup mode [ms]:"
    Textfield (211,326 104x30), "%6.1f", tooltip "Defines how often measurements will be taken and written to a file. Lower values will increase the file size.", text variable: GVL_Parameter.tMeas_ProductionMode
        OnMouseClick: write GVL_Parameter.tMeas_ProductionMode via Edit, min 10, max 100000, format 1000
    Label (15,325 185x30), "Meas. cycle Prod. mode [ms]:"
    Label (67,262 150x30), "Measurement frequency:"
END_VISUALIZATION

// ---- VISUs/MainWindow.TcVIS
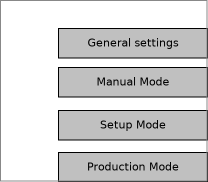
VISUALIZATION MainWindow  // 208x182
    Rectangle (58,152 150x30), "Production Mode", tooltip "Operation mode supposed to be used for production with slightly reduced measurement frequency."
        OnMouseClick: change screen: Production_Mode
    Rectangle (58,110 150x30), "Setup Mode", tooltip "Operation mode with increased measuring frequency in order to fine tune the process (e.g. reference values) according to your needs."
        OnMouseClick: change screen: Setup_Mode
    Rectangle (58,67 150x30), "Manual Mode", tooltip "Allows manual control (start/stop) of each and every subsystem."
        OnMouseClick: change screen: Manual_Mode
    Rectangle (58,28 150x30), "General settings", tooltip "Allows to adjust general system parameters, which will be applied in all different modes of operation."
        OnMouseClick: change screen: GeneralSettings
END_VISUALIZATION

// ---- VISUs/Manual_Mode.TcVIS
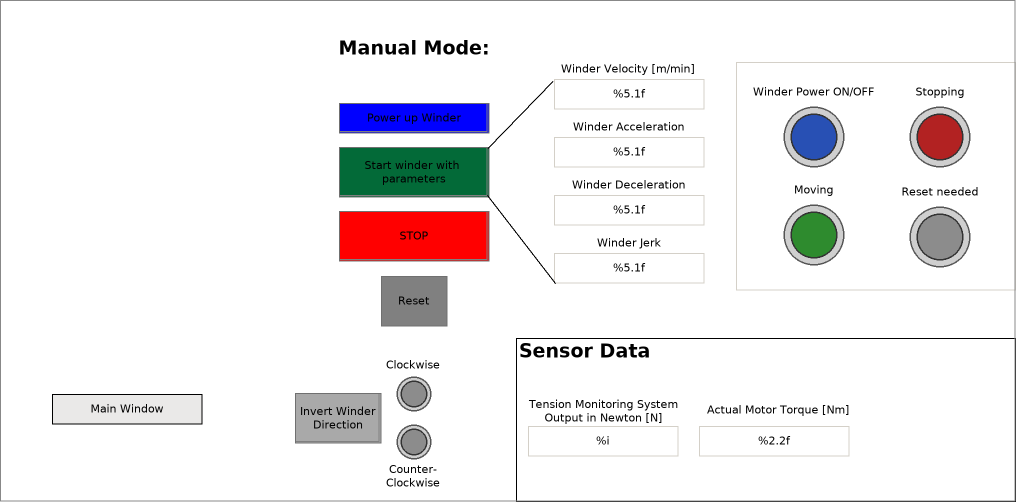
VISUALIZATION Manual_Mode  // 1016x502
    Rectangle (52,394 150x30), "Main Window"
        OnMouseClick: change screen: MainWindow
    Textfield (736,62 280x228)
    Textfield (516,338 500x164), "Sensor Data"
    Label (328,33 172x30), "Manual Mode:"
    Textfield (554,79 150x30), "%5.1f", text variable: GVL_Axis.rWinderVelocity
        OnMouseClick: write the text variable via VisuDialogs.Numpad, min 2.7, max 15
    Label (553,54 150x30), "Winder Velocity [m/min]"
    Textfield (554,137 150x30), "%5.1f", text variable: GVL_Axis.rWinderAcceleration
        OnMouseClick: write the text variable via Default
    Label (554,112 150x30), "Winder Acceleration"
    Textfield (554,253 150x30), "%5.1f", text variable: GVL_Axis.rWinderJerk
        OnMouseClick: write the text variable via Default
    Textfield (554,195 150x30), "%5.1f", text variable: GVL_Axis.rWinderDeceleration
        OnMouseClick: write the text variable via Default
    Label (554,170 150x30), "Winder Deceleration"
    Label (554,228 150x30), "Winder Jerk"
    Button (339,103 150x30), "Power up Winder", colour toggle: GVL_HMI.bButtonWinderPower
        toggle GVL_HMI.bButtonWinderPower
    Button (339,147 150x50), "Start winder with parameters", colour toggle: GVL_HMI.bButtonStartWinder
        OnMouseDown: execute { GVL_HMI.bButtonStartWinder := TRUE; }
        OnMouseUp: execute { GVL_HMI.bButtonStartWinder := FALSE; }
    Button (339,211 150x50), "STOP", colour toggle: GVL_HMI.bButtonStopWinder
        OnMouseDown: execute { GVL_HMI.bButtonStopWinder := TRUE; }
        OnMouseUp: execute { GVL_HMI.bButtonStopWinder := FALSE; }
    Button (381,276 66x50), "Reset", colour toggle: GVL_HMI.bButtonResetWinder
        OnMouseDown: execute { GVL_HMI.bButtonResetWinder := TRUE; }
        OnMouseUp: execute { GVL_HMI.bButtonResetWinder := FALSE; }
    Line (488,148) (553,81)
    Line (487,195) (555,283)
    Lamp1 (779,102 70x70), variable: GVL_Axis.bStatusPower, style: Lamp-Lamp1-Blue
    Label (739,77 150x30), "Winder Power ON/OFF"
    Lamp1 (779,200 70x70), variable: GVL_Axis.bStateCM, style: Lamp-Lamp1-Green
    Label (739,175 150x30), "Moving"
    Group (865,77 150x195)
        Lamp1 (40,25 70x70), variable: GVL_Axis.bStateStopping, style: Lamp-Lamp1-Red
        Label (0,0 150x30), "Stopping"
        Lamp1 (40,125 70x70), variable: GVL_Axis.bStateErrorStop, style: Lamp-Lamp1-Gray
        Label (0,100 150x30), "Reset needed"
    Textfield (528,426 150x30), "%i", text variable: GVL.iTensionMonitoringData
    Label (522,396 163x30), "Tension Monitoring System Output in Newton [N]"
    Button (295,393 86x50), "Invert Winder Direction", colour toggle: GVL_HMI.bButtonWinderDirection
        toggle GVL_HMI.bButtonWinderDirection
    Lamp1 (394,374 40x40), variable: GVL_HMI.bButtonWinderDirection, style: Lamp-Lamp1-Gray
    Lamp1 (394,422 40x40), variable: GVL_HMI.bButtonNotWinderDirection, style: Lamp-Lamp1-Gray
    Label (371,350 84x30), "Clockwise"
    Label (371,461 84x30), "Counter- Clockwise"
    Textfield (699,426 150x30), "%2.2f", text variable: GVL_HMI.ActTorque
    Label (697,395 163x30), "Actual Motor Torque [Nm]"
END_VISUALIZATION

// ---- VISUs/Production_Mode.TcVIS
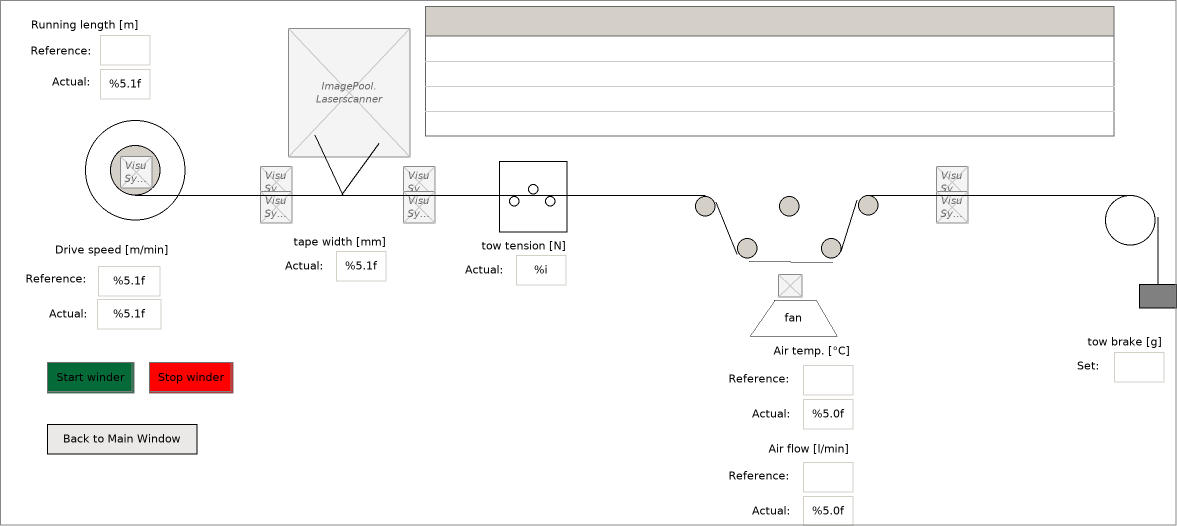
VISUALIZATION Production_Mode  // 1177x526
    Label (10,10 150x30), "Running length [m]"
    Textfield (100,35 50x30)
    Label (37,235 150x30), "Drive speed [m/min]"
    Textfield (97,299 64x30), "%5.1f", text variable: GVL_HMI.ActTapeSpeed
        OnMouseClick: write the text variable via Default
    Label (14,36 80x30), "Reference:"
    Label (13,67 80x30), "Actual:"
    Ellipse (85,120 100x100)
    Ellipse (110,145 50x50)
    Label (10,299 80x30), "Actual:"
    Label (9,264 80x30), "Reference:"
    Image (260,166 32x32), image: VisuSymbols.Symbols.TriangleDown
    Image (260,191 32x32), image: VisuSymbols.Symbols.TriangleUp
    Image (403,166 32x32), image: VisuSymbols.Symbols.TriangleDown
    Image (403,191 32x32), image: VisuSymbols.Symbols.TriangleUp
    Ellipse (695,196 20x20)
    Ellipse (737,238 20x20)
    Ellipse (779,196 20x20)
    Ellipse (821,238 20x20)
    Ellipse (858,195 20x20)
    Image (936,166 32x32), image: VisuSymbols.Symbols.TriangleDown
    Image (936,191 32x32), image: VisuSymbols.Symbols.TriangleUp
    Label (753,336 100x30), "Air temp. [°C]"
    Textfield (803,399 50x30), "%5.0f", text variable: GVL_Axis.rWinderVelocity
        OnMouseClick: write the text variable via Default
    Textfield (803,365 50x30)
    Label (713,399 80x30), "Actual:"
    Label (712,364 80x30), "Reference:"
    Label (752,434 100x30), "Air flow [l/min]"
    Textfield (803,496 50x30), "%5.0f", text variable: GVL_Axis.rWinderVelocity
        OnMouseClick: write the text variable via Default
    Textfield (803,462 50x30)
    Label (713,496 80x30), "Actual:"
    Label (712,461 80x30), "Reference:"
    Label (275,227 114x30), "tape width [mm]"
    Textfield (336,251 50x30), "%5.1f", text variable: GVL_Axis.rWinderVelocity
        OnMouseClick: write the text variable via Default
    Label (246,251 80x30), "Actual:"
    Polygon (775,300) (774,300) (816,300) (837,336) (750,336), "fan"
    Image (778,274 24x23), image: VisuSymbols.Symbols.ArrowBoldUp
    Line (737,254) (716,202)
    Line (749,261) (832,262)
    Label (455,231 114x30), "tow tension [N]"
    Textfield (516,255 50x30), "%i", text variable: GVL.iTensionMonitoringData
        OnMouseClick: write the text variable via Default
    Label (426,255 80x30), "Actual:"
    Label (1051,327 114x30), "tow brake [g]"
    Label (1022,351 80x30), "Set:"
    Textfield (1114,352 50x30)
    Table (425,6 689x130), data array: GVL.LaserScannerData
        p3854506369: GVL.LaserScannerData[INDEX]
    Rectangle (47,424 150x30), "Back to Main Window"
        OnMouseClick: change screen: MainWindow
    Textfield (100,69 50x30), "%5.1f", text variable: GVL_HMI.RunningLength
        OnMouseClick: write the text variable via Default
    Rectangle (499,161 68x71)
    Ellipse (509,196 10x10)
    Ellipse (528,184 10x10)
    Ellipse (545,196 10x10)
    Line (135,195) (705,195)
    Line (841,251) (857,200)
    Line (867,195) (1132,195)
    Ellipse (1105,195 50x50)
    Line (1158,288) (1158,217)
    Rectangle (1139,284 38x24)
    Image (288,28 122x129), image: ImagePool.Laserscanner
    Line (342,194) (379,143)
    Line (343,195) (315,135)
    Textfield (98,266 62x30), "%5.1f", text variable: GVL_Axis.rWinderVelocity
        OnMouseClick: write the text variable via VisuDialogs.Numpad, min 2.7, max 15
    Button (47,362 87x31), "Start winder", colour toggle: GVL_HMI.bButtonStartWinder
        OnMouseDown: execute { GVL_HMI.bButtonStartWinder := TRUE; }
        OnMouseUp: execute { GVL_HMI.bButtonStartWinder := FALSE; }
    Button (149,362 84x31), "Stop winder", colour toggle: GVL_HMI.bButtonStopWinder
        OnMouseDown: execute { GVL_HMI.bButtonStopWinder := TRUE; }
        OnMouseUp: execute { GVL_HMI.bButtonStopWinder := FALSE; }
    Image (120,156 32x32), image: VisuSymbols.Symbols.ArrowHalfRightUp
END_VISUALIZATION

// ---- VISUs/Setup_Mode.TcVIS
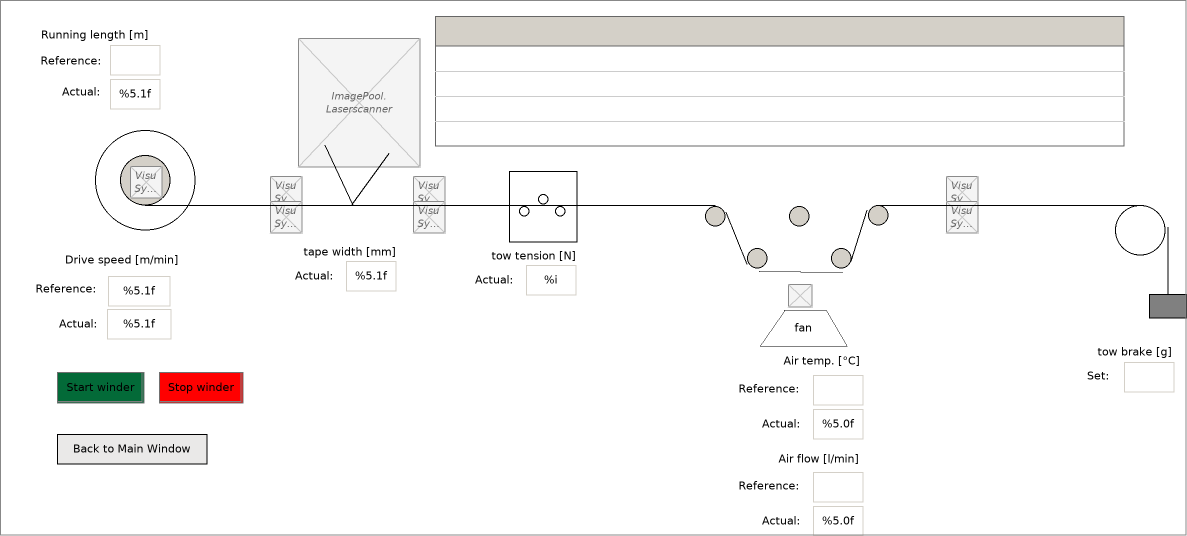
VISUALIZATION Setup_Mode  // 1187x536
    Label (20,20 150x30), "Running length [m]"
    Textfield (110,45 50x30)
    Label (47,245 150x30), "Drive speed [m/min]"
    Textfield (107,309 64x30), "%5.1f", text variable: GVL_HMI.ActTapeSpeed
        OnMouseClick: write the text variable via Default
    Label (24,46 80x30), "Reference:"
    Label (23,77 80x30), "Actual:"
    Ellipse (95,130 100x100)
    Ellipse (120,155 50x50)
    Label (20,309 80x30), "Actual:"
    Label (19,274 80x30), "Reference:"
    Image (270,176 32x32), image: VisuSymbols.Symbols.TriangleDown
    Image (270,201 32x32), image: VisuSymbols.Symbols.TriangleUp
    Image (413,176 32x32), image: VisuSymbols.Symbols.TriangleDown
    Image (413,201 32x32), image: VisuSymbols.Symbols.TriangleUp
    Ellipse (705,206 20x20)
    Ellipse (747,248 20x20)
    Ellipse (789,206 20x20)
    Ellipse (831,248 20x20)
    Ellipse (868,205 20x20)
    Image (946,176 32x32), image: VisuSymbols.Symbols.TriangleDown
    Image (946,201 32x32), image: VisuSymbols.Symbols.TriangleUp
    Label (763,346 100x30), "Air temp. [°C]"
    Textfield (813,409 50x30), "%5.0f", text variable: GVL_Axis.rWinderVelocity
        OnMouseClick: write the text variable via Default
    Textfield (813,375 50x30)
    Label (723,409 80x30), "Actual:"
    Label (722,374 80x30), "Reference:"
    Label (762,444 100x30), "Air flow [l/min]"
    Textfield (813,506 50x30), "%5.0f", text variable: GVL_Axis.rWinderVelocity
        OnMouseClick: write the text variable via Default
    Textfield (813,472 50x30)
    Label (723,506 80x30), "Actual:"
    Label (722,471 80x30), "Reference:"
    Label (285,237 114x30), "tape width [mm]"
    Textfield (346,261 50x30), "%5.1f", text variable: GVL_Axis.rWinderVelocity
        OnMouseClick: write the text variable via Default
    Label (256,261 80x30), "Actual:"
    Polygon (785,310) (784,310) (826,310) (847,346) (760,346), "fan"
    Image (788,284 24x23), image: VisuSymbols.Symbols.ArrowBoldUp
    Line (747,264) (726,212)
    Line (759,271) (842,272)
    Label (465,241 114x30), "tow tension [N]"
    Textfield (526,265 50x30), "%i", text variable: GVL.iTensionMonitoringData
        OnMouseClick: write the text variable via Default
    Label (436,265 80x30), "Actual:"
    Label (1061,337 114x30), "tow brake [g]"
    Label (1032,361 80x30), "Set:"
    Textfield (1124,362 50x30)
    Table (435,16 689x130), data array: GVL.LaserScannerData
        p3854506369: GVL.LaserScannerData[INDEX]
    Rectangle (57,434 150x30), "Back to Main Window"
        OnMouseClick: change screen: MainWindow
    Textfield (110,79 50x30), "%5.1f", text variable: GVL_HMI.RunningLength
        OnMouseClick: write the text variable via Default
    Rectangle (509,171 68x71)
    Ellipse (519,206 10x10)
    Ellipse (538,194 10x10)
    Ellipse (555,206 10x10)
    Line (145,205) (715,205)
    Line (851,261) (867,210)
    Line (877,205) (1142,205)
    Ellipse (1115,205 50x50)
    Line (1168,298) (1168,227)
    Rectangle (1149,294 38x24)
    Image (298,38 122x129), image: ImagePool.Laserscanner
    Line (352,204) (389,153)
    Line (353,205) (325,145)
    Textfield (108,276 62x30), "%5.1f", text variable: GVL_Axis.rWinderVelocity
        OnMouseClick: write the text variable via VisuDialogs.Numpad, min 2.7, max 15
    Button (57,372 87x31), "Start winder", colour toggle: GVL_HMI.bButtonStartWinder
        OnMouseDown: execute { GVL_HMI.bButtonStartWinder := TRUE; }
        OnMouseUp: execute { GVL_HMI.bButtonStartWinder := FALSE; }
    Button (159,372 84x31), "Stop winder", colour toggle: GVL_HMI.bButtonStopWinder
        OnMouseDown: execute { GVL_HMI.bButtonStopWinder := TRUE; }
        OnMouseUp: execute { GVL_HMI.bButtonStopWinder := FALSE; }
    Image (130,166 32x32), image: VisuSymbols.Symbols.ArrowHalfRightUp
END_VISUALIZATION

// ---- VISUs/Winder_control.TcVIS
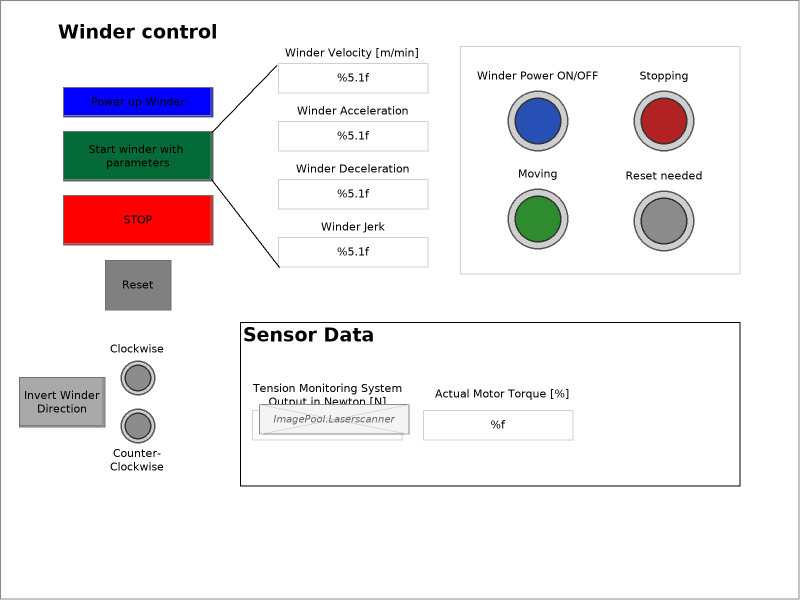
VISUALIZATION Winder_control  // 800x600
    Textfield (460,46 280x228)
    Textfield (240,322 500x164), "Sensor Data"
    Label (52,17 172x30), "Winder control"
    Textfield (278,63 150x30), "%5.1f", text variable: GVL_Axis.rWinderVelocity
        OnMouseClick: write the text variable via VisuDialogs.Numpad, min 2.7, max 15
    Label (277,38 150x30), "Winder Velocity [m/min]"
    Textfield (278,121 150x30), "%5.1f", text variable: GVL_Axis.rWinderAcceleration
        OnMouseClick: write the text variable via Default
    Label (278,96 150x30), "Winder Acceleration"
    Textfield (278,237 150x30), "%5.1f", text variable: GVL_Axis.rWinderJerk
        OnMouseClick: write the text variable via Default
    Textfield (278,179 150x30), "%5.1f", text variable: GVL_Axis.rWinderDeceleration
        OnMouseClick: write the text variable via Default
    Label (278,154 150x30), "Winder Deceleration"
    Label (278,212 150x30), "Winder Jerk"
    Button (63,87 150x30), "Power up Winder", colour toggle: GVL_HMI.bButtonWinderPower
        toggle GVL_HMI.bButtonWinderPower
    Button (63,131 150x50), "Start winder with parameters", colour toggle: GVL_HMI.bButtonStartWinder
        OnMouseDown: execute { GVL_HMI.bButtonStartWinder := TRUE; }
        OnMouseUp: execute { GVL_HMI.bButtonStartWinder := FALSE; }
    Button (63,195 150x50), "STOP", colour toggle: GVL_HMI.bButtonStopWinder
        OnMouseDown: execute { GVL_HMI.bButtonStopWinder := TRUE; }
        OnMouseUp: execute { GVL_HMI.bButtonStopWinder := FALSE; }
    Button (105,260 66x50), "Reset", colour toggle: GVL_HMI.bButtonResetWinder
        OnMouseDown: execute { GVL_HMI.bButtonResetWinder := TRUE; }
        OnMouseUp: execute { GVL_HMI.bButtonResetWinder := FALSE; }
    Line (212,132) (277,65)
    Line (211,179) (279,267)
    Lamp1 (503,86 70x70), variable: GVL_Axis.bStatusPower, style: Lamp-Lamp1-Blue
    Label (463,61 150x30), "Winder Power ON/OFF"
    Lamp1 (503,184 70x70), variable: GVL_Axis.bStateCM, style: Lamp-Lamp1-Green
    Label (463,159 150x30), "Moving"
    Group (589,61 150x195)
        Lamp1 (40,25 70x70), variable: GVL_Axis.bStateStopping, style: Lamp-Lamp1-Red
        Label (0,0 150x30), "Stopping"
        Lamp1 (40,125 70x70), variable: GVL_Axis.bStateErrorStop, style: Lamp-Lamp1-Gray
        Label (0,100 150x30), "Reset needed"
    Textfield (252,410 150x30), "%i", text variable: GVL.iTensionMonitoringData
    Label (246,380 163x30), "Tension Monitoring System Output in Newton [N]"
    Button (19,377 86x50), "Invert Winder Direction", colour toggle: GVL_HMI.bButtonWinderDirection
        toggle GVL_HMI.bButtonWinderDirection
    Lamp1 (118,358 40x40), variable: GVL_HMI.bButtonWinderDirection, style: Lamp-Lamp1-Gray
    Lamp1 (118,406 40x40), variable: GVL_HMI.bButtonNotWinderDirection, style: Lamp-Lamp1-Gray
    Label (95,334 84x30), "Clockwise"
    Label (95,445 84x30), "Counter- Clockwise"
    Textfield (237,275 231x45), "!!New Motion Parameter detected!! Click 'Start winder' to update Parameters", colour toggle: GVL_Axis.bNewMotionParameter
    Textfield (423,410 150x30), "%f", text variable: GVL_HMI.ActTorque
    Label (421,379 163x30), "Actual Motor Torque [%]"
    Image (259,404 150x30), image: ImagePool.Laserscanner
END_VISUALIZATION
